FUNCTION WStrConcat : WSTRING(511)
VAR_INPUT
	str0 : WSTRING(511) := "";
	str1 : WSTRING(511) := "";
	str2 : WSTRING(511) := "";
	str3 : WSTRING(511) := "";
	str4 : WSTRING(511) := "";
	str5 : WSTRING(511) := "";
	str6 : WSTRING(511) := "";
	str7 : WSTRING(511) := "";
	str8 : WSTRING(511) := "";
END_VAR
VAR
	tmpstr : WSTRING(511);
END_VAR

tmpstr := WCONCAT(STR1:= str0, STR2:= str1);
tmpstr := WCONCAT(STR1:= tmpstr, STR2:= str2);
tmpstr := WCONCAT(STR1:= tmpstr, STR2:= str3);
tmpstr := WCONCAT(STR1:= tmpstr, STR2:= str4);
tmpstr := WCONCAT(STR1:= tmpstr, STR2:= str5);
tmpstr := WCONCAT(STR1:= tmpstr, STR2:= str6);
tmpstr := WCONCAT(STR1:= tmpstr, STR2:= str7);
tmpstr := WCONCAT(STR1:= tmpstr, STR2:= str8);
WStrConcat := tmpstr;
RETURN;

END_FUNCTION

(* stored: Version 1.1.0.1, ProductVersion 3.1.4026.13
   POU WStrConcat: Id {8adb4079-c139-41a2-89e4-160e3112ca3f}, SpecialFunc None *)
